(* LS Electric XG5000 project: IEC164S *)
(* PLC LSPLC *)

PROGRAM NewProgram (* task: 스캔 프로그램 *)

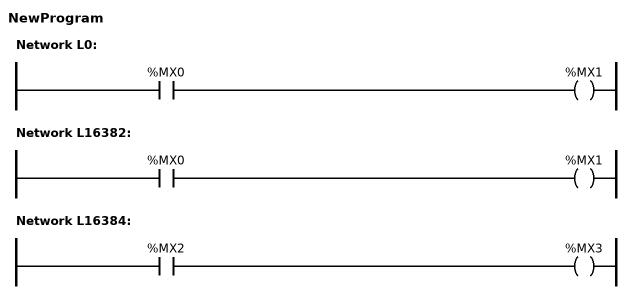
(* Rung L0 *)
%MX1 := %MX0;
(* Rung L16382 *)
%MX1 := %MX0;
(* Rung L16384 *)
%MX3 := %MX2;
END_PROGRAM